// TIA Portal V18 export
DATA_BLOCK "valve_DB"   // DB116
VERSION : 0.1
// stored: AutoNumber true, DBAccessibleFromOPCUA true, DBAccessibleFromWebserver true, InstanceOfName valve, InstanceOfType FB
"valve"
   // VAR_INPUT
   //    "A/M" : Bool;
   //    open_auto : Bool;
   //    open_man : Bool;
   //    fbk_open : Bool;
   //    fbk_close : Bool;
   //    reset : Bool;
   //    intl : Bool;
   //    Mon_En : Bool;
   //    mon_sp : Time;
   //    run_fb : Bool;
   //    stop_fb : Bool;
   // END_VAR
   // VAR_OUTPUT
   //    "open/close" : Bool;
   //    fault : Bool;
   //    status : Int;
   // END_VAR
   // VAR
   //    open_fault : Bool;
   //    close_fault : Bool;
   //    IEC_Timer_0_Instance { S7_SetPoint := 'True'} : TON_TIME;
   //    IEC_Timer_0_Instance_1 { S7_SetPoint := 'True'} : TON_TIME;
   //    mon : Int;
   //    pulse : Bool;
   //    pulse1 : Bool;
   //    mon1 : Int;
   //    IEC_Timer_0_Instance_2 { S7_SetPoint := 'True'} : TON_TIME;
   // END_VAR
BEGIN
END_DATA_BLOCK
